KUKA KRL program: Rack_Verde_Inpicker_D.src, Rack_Verde_Inpicker_D.dat

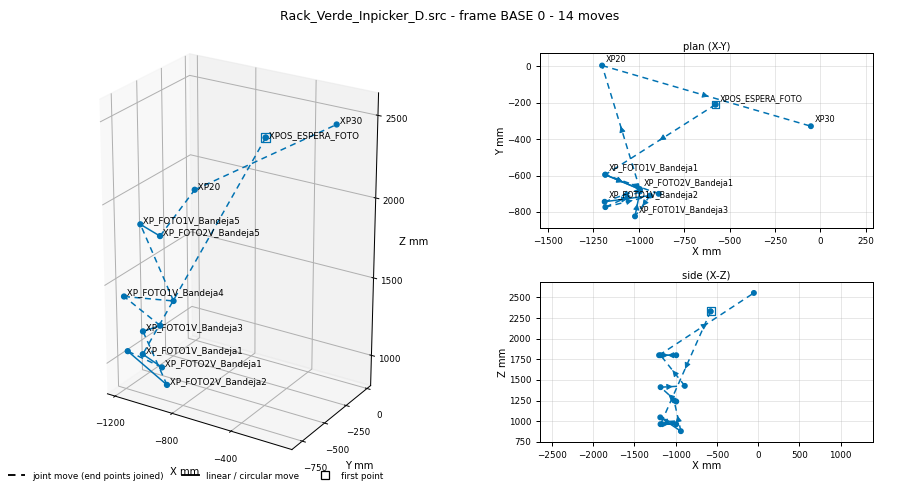
[picture p0: tool path of Rack_Verde_Inpicker_D.src in frame BASE 0, 14 of 14 moves have a stored position in this frame; points joined in program order, loops and branches not executed]
--- Rack_Verde_Inpicker_D.src ---
&ACCESS RVP
&REL 1
&COMMENT FOTOS EN RACK VERDE
&PARAM EDITMASK = *
&PARAM TEMPLATE = C:\KRC\Roboter\Template\vorgabe
&PARAM DISKPATH = KRC:\R1\Program\MAFELEC
DEF Rack_Verde_Inpicker_D( )
;FOLD DECLARACION_INPICKER
DECL EKI_STATUS Ret
DECL INT InPickerStateValue
;ENDFOLD
;FOLD INI;%{PE}
  ;FOLD BASISTECH INI
    GLOBAL INTERRUPT DECL 3 WHEN $STOPMESS==TRUE DO IR_STOPM ( )
    INTERRUPT ON 3
    BAS (#INITMOV,0 )
  ;ENDFOLD (BASISTECH INI)
  ;FOLD USER INI
O_LIMITS_OK=FALSE
O_LIMITS_NOK=FALSE
O_LIMIT_X=FALSE
O_LIMIT_Y=FALSE
O_LIMIT_Z=FALSE
O_LIMIT_A=FALSE
O_LIMIT_B=FALSE
O_LIMIT_C=FALSE
LIM_X=FALSE
LIM_Y=FALSE
LIM_Z=FALSE
LIM_A=FALSE
LIM_B=FALSE
LIM_C=FALSE
O_TYPE_INFO=0

  ;ENDFOLD (USER INI)
;ENDFOLD (INI)

;################################################
; PROYECTO: MAFELEC PLANTA DE BATERIAS
; ROBOT: 121_R1
; PROGRAMA: FOTO PARA CORRECCIONES EN RACK VERDE
; CREADO POR: Alejandro Company(zaisor robotics)
; FECHA: 23-NOVIEMBRE-2022
; MODIFICADO POR:
; FECHA MODIFICACION: 13-ENERO-2023
;################################################

$TIMER[2]=0
$TIMER_STOP[2]=FALSE
;FOLD INICIALIZACION PUERTOS DE KRL
Ret = EKI_INIT("XML_Kuka_InPicker_1")
Ret = EKI_INIT("XML_Kuka_InPicker_2")

Ret = EKI_OPEN("XML_Kuka_InPicker_1")
Ret = EKI_OPEN("XML_Kuka_InPicker_2")

 INPICKER_Handler.DataToSend.command=0
;WAIT FOR (INPICKER_Handler.ConnectionStatus==TRUE)
;IF (INPICKER_Handler.ConnectionStatus==TRUE) THEN
;ELSE
;ENDIF

;ENDFOLD

Empujador(1,"R",FALSE)
Empujador(2,"R",FALSE)

; POSICION DE ESPERA ENTRADA RACK 1
;FOLD PTP POS_ESPERA_FOTO Vel=100 % H Tool[5]:T_Camara Base[0];%{PE}%R 8.3.48,%MKUKATPBASIS,%CMOVE,%VPTP,%P 1:PTP, 2:POS_ESPERA_FOTO, 3:, 5:100, 7:H
$BWDSTART=FALSE
PDAT_ACT=PH
FDAT_ACT=FPOS_ESPERA_FOTO
BAS(#PTP_PARAMS,100)
PTP XPOS_ESPERA_FOTO
;ENDFOLD

;ESPERA AREA 1
WAIT FOR I_ARDY_1
O_AREL_1=FALSE
RV_Bandeja_nr=0

Empujador(1,"R",TRUE)
Empujador(2,"R",TRUE)

;FOLD PTP P11 CONT Vel=100 % M Tool[5]:T_Camara Base[0];%{PE}%R 8.3.48,%MKUKATPBASIS,%CMOVE,%VPTP,%P 1:PTP, 2:P11, 3:C_DIS, 5:100, 7:M
$BWDSTART=FALSE
PDAT_ACT=PM
FDAT_ACT=FP11
BAS(#PTP_PARAMS,100)
PTP XP11 C_DIS
;ENDFOLD

O_TYPE_RQ=TRUE
WAIT FOR (I_TYPE_INFO >= 10) AND (I_TYPE_INFO <= 16)

RV_Bandeja_Nr=I_TYPE_INFO

SWITCH RV_Bandeja_Nr

CASE 11
O_TYPE_RQ=FALSE
O_TYPE_INFO=RV_Bandeja_Nr
INICIO_FOTO1:
;FOLD PTP P_FOTO1V_Bandeja1 Vel=50 % M Tool[5]:T_Camara Base[0];%{PE}%R 8.3.48,%MKUKATPBASIS,%CMOVE,%VPTP,%P 1:PTP, 2:P_FOTO1V_Bandeja1, 3:, 5:50, 7:M
$BWDSTART=FALSE
PDAT_ACT=PM
FDAT_ACT=FP_FOTO1V_Bandeja1
BAS(#PTP_PARAMS,50)
PTP XP_FOTO1V_Bandeja1
;ENDFOLD
;FOLD REALIZA FOTO 1 BANDEJA 1
WAIT SEC 1
Fallo_nr=0
Ini1:
O_INPICKER_OK = FALSE
O_INPICKER_NOK = FALSE
SELECT_SIN=FALSE
SELECT_U1=FALSE
SELECT_U2=FALSE
SELECT_U3=FALSE
SELECT_U4=FALSE

; INICIALIZACION CAMARA PARA BANDEJA 1
 INPICKER_Handler.DataToSend.command=0
 INPICKER_Handler.DataToSend.GraspConfirmation=0
 WAIT FOR (INPICKER_Handler.DataReceived.state==0)

; Camara siempre 2
 INPICKER_Handler.DataToSend.CameraID=2

; contendor igual al numero de bandeja
 INPICKER_Handler.DataToSend.ContainerID=1
 INPICKER_Handler.DataToSend.partid=1
 INPICKER_Handler.DataToSend.GraspConfirmation=0
 WAIT SEC 0.2

; DISPARO FOTO
 INPICKER_Handler.DataToSend.command=1

; ESPERA FOTO REALIZADA
 WAIT FOR (INPICKER_Handler.DataReceived.state==15) OR (INPICKER_Handler.DataReceived.state==-1)

IF (INPICKER_Handler.DataReceived.state==-1) THEN

IF (Fallo_nr>=1) THEN
O_INPICKER_OK=FALSE
O_INPICKER_NOK=TRUE

O_TYPE_RQ = FALSE
WAIT FOR I_TYPE_INFO == 0

O_TYPE_RQ = TRUE
WAIT FOR (I_TYPE_INFO >= 1) AND (I_TYPE_INFO <= 5)

SWITCH I_TYPE_INFO

CASE 2
; #### SELECCION DESDE HMI REINTENTO FOTO ####

SELECT_NEXT=FALSE
O_INPICKER_OK=FALSE
O_INPICKER_NOK=FALSE
O_TYPE_RQ = FALSE
GOTO Ini1

CASE 3
; #### SELECCION DESDE HMI CONT SIN CORRECCION ####

SELECT_SIN=TRUE
O_INPICKER_OK=FALSE
O_INPICKER_NOK=TRUE
O_TYPE_RQ = FALSE
GOTO FIN_FOTO1

CASE 4
; #### SELECCION DESDE HMI CERRAR BANDEJA ####
; #### E IR A SIGUIENTE NIVEL             ####

SELECT_NEXT=TRUE
O_INPICKER_OK=FALSE
O_INPICKER_NOK=FALSE
O_TYPE_RQ = FALSE
GOTO FIN_FOTO1

DEFAULT
ENDSWITCH

ELSE

Fallo_nr=Fallo_nr+1
GOTO Ini1

ENDIF
ENDIF

Fin1:
 WAIT SEC 0.1
;ENDFOLD

INICIO_POS2_B1:
;FOLD LIN P_FOTO2V_Bandeja1 Vel=0.5 m/s M Tool[5]:T_Camara Base[0];%{PE}%R 8.3.48,%MKUKATPBASIS,%CMOVE,%VLIN,%P 1:LIN, 2:P_FOTO2V_Bandeja1, 3:, 5:0.5, 7:M
$BWDSTART=FALSE
LDAT_ACT=LM
FDAT_ACT=FP_FOTO2V_Bandeja1
BAS(#CP_PARAMS,0.5)
LIN XP_FOTO2V_Bandeja1
;ENDFOLD
;FOLD REALIZA FOTO 2 BANDEJA 1 (INFERIOR)
WAIT SEC 1.0
INPICKER_Handler.DataToSend.GraspConfirmation=1

WAIT FOR (INPICKER_Handler.DataReceived.state==30) OR (INPICKER_Handler.dataReceived.state==-1)

WAIT SEC 0.5

INPICKER_Handler.DataToSend.command=0

IF (INPICKER_handler.datareceived.state==30 ) THEN

IF (INPICKER_Handler.DataReceived.ObjectsGraspable>0) THEN

O_INPICKER_OK=TRUE
O_INPICKER_NOK=FALSE

ELSE

O_INPICKER_OK=FALSE
O_INPICKER_NOK=TRUE

ENDIF

ENDIF

IF (INPICKER_handler.datareceived.state==-1 ) OR (INPICKER_Handler.DataReceived.ObjectsGraspable<=0) THEN

O_INPICKER_OK=FALSE
O_INPICKER_NOK=TRUE

O_TYPE_RQ = FALSE
WAIT FOR I_TYPE_INFO == 0

O_TYPE_RQ = TRUE
WAIT FOR (I_TYPE_INFO >= 1) AND (I_TYPE_INFO <= 5)

SWITCH I_TYPE_INFO

CASE 2
; #### SELECCION DESDE HMI REINTENTO FOTO ####

SELECT_NEXT=FALSE
O_INPICKER_OK=FALSE
O_INPICKER_NOK=FALSE
O_TYPE_RQ = FALSE

IF (INPICKER_Handler.DataReceived.ObjectsGraspable>0)THEN
ELSE
GOTO INICIO_FOTO1
ENDIF

WAIT FOR (INPICKER_Handler.DataReceived.state==0)
GOTO INICIO_FOTO1

CASE 3
; #### SELECCION DESDE HMI CONT SIN CORRECCION ####

SELECT_NEXT=FALSE
O_TYPE_RQ = FALSE

CASE 4
; #### SELECCION DESDE HMI CERRAR BANDEJA ####
; #### E IR A SIGUIENTE NIVEL             ####

SELECT_NEXT=TRUE
O_INPICKER_OK=FALSE
O_INPICKER_NOK=FALSE
O_TYPE_RQ = FALSE

DEFAULT
ENDSWITCH

ENDIF
 INPICKER_Handler.DataToSend.command=0

;ENDFOLD
;FOLD ACTUALIZA BASE DE DESCARGA
FRAMEAUX={X 0,Y 0,Z 0,A 0,B 0,C 0}
FRAME_POS={X 0,Y 0,Z 0,A 0,B 0,C 0}

FRAMEAUX=INPICKER_Handler.DataReceived.PartsToGrasp0.Position
FRAME_POS.x=(FRAMEAUX.x/10)
FRAME_POS.y=(FRAMEAUX.y/10)
FRAME_POS.z=(FRAMEAUX.z/10)
FRAME_POS.a=(FRAMEAUX.a/10)
FRAME_POS.b=(FRAMEAUX.b/10)
FRAME_POS.c=(FRAMEAUX.c/10)

IF FRAME_POS.A < 180.0 THEN
FRAME_POS.A = FRAME_POS.A + 360
ENDIF
IF FRAME_POS.B < 180.0 THEN
FRAME_POS.B = FRAME_POS.B + 360
ENDIF
IF FRAME_POS.A > 180.0 THEN
FRAME_POS.A = FRAME_POS.A - 360
ENDIF
IF FRAME_POS.B > 180.0 THEN
FRAME_POS.B = FRAME_POS.B - 360
ENDIF

FRAME_POS.C = FRAME_POS.C - 360

;ENDFOLD
;FOLD CONTROL LIMITES DE VISION
CTRL_limites()
;ENDFOLD
;FOLD DECISION RESULTADOS EVALUACION BANDEJA 1
IF (O_LIMITS_OK==FALSE) AND (O_LIMITS_NOK==TRUE) THEN

O_TYPE_RQ = FALSE
WAIT FOR I_TYPE_INFO == 0

O_TYPE_RQ = TRUE
WAIT FOR (I_TYPE_INFO >= 1) AND (I_TYPE_INFO <= 5)

SWITCH I_TYPE_INFO

CASE 2
; #### SELECCION DESDE HMI REINTENTO FOTO ####

SELECT_NEXT=FALSE
O_TYPE_RQ = FALSE
O_LIMITS_OK = FALSE
O_LIMITS_NOK = FALSE
O_LIMIT_X = FALSE
O_LIMIT_Y = FALSE
O_LIMIT_Z = FALSE
O_LIMIT_A = FALSE
O_LIMIT_B = FALSE
O_LIMIT_C = FALSE

GOTO INICIO_FOTO1

CASE 3
; #### SELECCION DESDE HMI CONT SIN CORRECCION ####

SELECT_NEXT=FALSE
O_TYPE_RQ = FALSE

CASE 4
; #### SELECCION DESDE HMI CERRAR BANDEJA ####
; #### E IR A SIGUIENTE NIVEL             ####

SELECT_NEXT=TRUE
O_TYPE_RQ = FALSE
O_LIMITS_OK = FALSE
O_LIMITS_NOK = FALSE
O_LIMIT_X = FALSE
O_LIMIT_Y = FALSE
O_LIMIT_Z = FALSE
O_LIMIT_A = FALSE
O_LIMIT_B = FALSE
O_LIMIT_C = FALSE

DEFAULT

HALT
HALT
HALT
ENDSWITCH

ENDIF
;ENDFOLD
FIN_FOTO1:

CASE 12
O_TYPE_RQ=FALSE
O_TYPE_INFO=RV_Bandeja_Nr
INICIO_FOTO2:
;FOLD PTP P_FOTO1V_Bandeja2 Vel=50 % M Tool[5]:T_Camara Base[0];%{PE}%R 8.3.48,%MKUKATPBASIS,%CMOVE,%VPTP,%P 1:PTP, 2:P_FOTO1V_Bandeja2, 3:, 5:50, 7:M
$BWDSTART=FALSE
PDAT_ACT=PM
FDAT_ACT=FP_FOTO1V_Bandeja2
BAS(#PTP_PARAMS,50)
PTP XP_FOTO1V_Bandeja2
;ENDFOLD
;FOLD REALIZA FOTO 1 BANDEJA 2
WAIT SEC 1
Fallo_nr=0
Ini2:
O_INPICKER_OK = FALSE
O_INPICKER_NOK = FALSE
SELECT_SIN=FALSE
SELECT_U1=FALSE
SELECT_U2=FALSE
SELECT_U3=FALSE
SELECT_U4=FALSE

; INICIALIZACION CAMARA PARA BANDEJA 2
 INPICKER_Handler.DataToSend.command=0
 INPICKER_Handler.DataToSend.GraspConfirmation=0
 WAIT FOR (INPICKER_Handler.DataReceived.state==0)

; Camara siempre 2
 INPICKER_Handler.DataToSend.CameraID=2

; contendor igual al numero de bandeja
 INPICKER_Handler.DataToSend.ContainerID=2
 INPICKER_Handler.DataToSend.partid=2
 INPICKER_Handler.DataToSend.GraspConfirmation=0
 WAIT SEC 0.2

; DISPARO FOTO
 INPICKER_Handler.DataToSend.command=1

; ESPERA FOTO REALIZADA
 WAIT FOR (INPICKER_Handler.DataReceived.state==15) OR (INPICKER_Handler.DataReceived.state==-1)

IF (INPICKER_Handler.DataReceived.state==-1) THEN

IF (Fallo_nr>=1) THEN
O_INPICKER_OK=FALSE
O_INPICKER_NOK=TRUE

O_TYPE_RQ = FALSE
WAIT FOR I_TYPE_INFO == 0

O_TYPE_RQ = TRUE
WAIT FOR (I_TYPE_INFO >= 1) AND (I_TYPE_INFO <= 5)

SWITCH I_TYPE_INFO

CASE 2
; #### SELECCION DESDE HMI REINTENTO FOTO ####

SELECT_NEXT=FALSE
O_INPICKER_OK=FALSE
O_INPICKER_NOK=FALSE
O_TYPE_RQ = FALSE
GOTO Ini2

CASE 3
; #### SELECCION DESDE HMI CONT SIN CORRECCION ####

SELECT_SIN=TRUE
O_INPICKER_OK=FALSE
O_INPICKER_NOK=TRUE
O_TYPE_RQ = FALSE
GOTO FIN_FOTO2

CASE 4
; #### SELECCION DESDE HMI CERRAR BANDEJA ####
; #### E IR A SIGUIENTE NIVEL             ####

SELECT_NEXT=TRUE
O_INPICKER_OK=FALSE
O_INPICKER_NOK=FALSE
O_TYPE_RQ = FALSE
GOTO FIN_FOTO2

DEFAULT
ENDSWITCH

ELSE

Fallo_nr=Fallo_nr+1
GOTO Ini2

ENDIF
ENDIF

Fin2:
 WAIT SEC 0.1
;ENDFOLD

INICIO_POS2_B2:
;FOLD LIN P_FOTO2V_Bandeja2 Vel=0.5 m/s M Tool[5]:T_Camara Base[0];%{PE}%R 8.3.48,%MKUKATPBASIS,%CMOVE,%VLIN,%P 1:LIN, 2:P_FOTO2V_Bandeja2, 3:, 5:0.5, 7:M
$BWDSTART=FALSE
LDAT_ACT=LM
FDAT_ACT=FP_FOTO2V_Bandeja2
BAS(#CP_PARAMS,0.5)
LIN XP_FOTO2V_Bandeja2
;ENDFOLD
;FOLD REALIZA FOTO 2 BANDEJA 2
WAIT SEC 1.0
INPICKER_Handler.DataToSend.GraspConfirmation=1

WAIT FOR (INPICKER_Handler.DataReceived.state==30) OR (INPICKER_Handler.dataReceived.state==-1)

WAIT SEC 0.5
INPICKER_Handler.DataToSend.command=0

IF (INPICKER_handler.datareceived.state==30 ) THEN

IF (INPICKER_Handler.DataReceived.ObjectsGraspable>0) THEN

O_INPICKER_OK=TRUE
O_INPICKER_NOK=FALSE

ELSE

O_INPICKER_OK=FALSE
O_INPICKER_NOK=TRUE

ENDIF

ENDIF

IF (INPICKER_handler.datareceived.state==-1 ) OR (INPICKER_Handler.DataReceived.ObjectsGraspable<=0) THEN

O_INPICKER_OK=FALSE
O_INPICKER_NOK=TRUE

O_TYPE_RQ = FALSE
WAIT FOR I_TYPE_INFO == 0

O_TYPE_RQ = TRUE
WAIT FOR (I_TYPE_INFO >= 1) AND (I_TYPE_INFO <= 5)

SWITCH I_TYPE_INFO

CASE 2
; #### SELECCION DESDE HMI REINTENTO FOTO ####

SELECT_NEXT=FALSE
O_INPICKER_OK=FALSE
O_INPICKER_NOK=FALSE
O_TYPE_RQ = FALSE

IF (INPICKER_Handler.DataReceived.ObjectsGraspable>0)THEN
ELSE
GOTO INICIO_FOTO2
ENDIF

WAIT FOR (INPICKER_Handler.DataReceived.state==0)
GOTO INICIO_FOTO2

CASE 3
; #### SELECCION DESDE HMI CONT SIN CORRECCION ####

SELECT_NEXT=FALSE
O_TYPE_RQ = FALSE

CASE 4
; #### SELECCION DESDE HMI CERRAR BANDEJA ####
; #### E IR A SIGUIENTE NIVEL             ####

SELECT_NEXT=TRUE
O_INPICKER_OK=FALSE
O_INPICKER_NOK=FALSE
O_TYPE_RQ = FALSE

DEFAULT
ENDSWITCH

ENDIF

 INPICKER_Handler.DataToSend.command=0

;ENDFOLD
;FOLD ACTUALIZA BASE DE DESCARGA
FRAMEAUX={X 0,Y 0,Z 0,A 0,B 0,C 0}
FRAME_POS={X 0,Y 0,Z 0,A 0,B 0,C 0}

FRAMEAUX=INPICKER_Handler.DataReceived.PartsToGrasp0.Position
FRAME_POS.x=(FRAMEAUX.x/10)
FRAME_POS.y=(FRAMEAUX.y/10)
FRAME_POS.z=(FRAMEAUX.z/10)
FRAME_POS.a=(FRAMEAUX.a/10)
FRAME_POS.b=(FRAMEAUX.b/10)
FRAME_POS.c=(FRAMEAUX.c/10)

IF FRAME_POS.A < 180.0 THEN
FRAME_POS.A = FRAME_POS.A + 360
ENDIF

IF FRAME_POS.B < 180.0 THEN
FRAME_POS.B = FRAME_POS.B + 360
ENDIF

IF FRAME_POS.A > 180.0 THEN
FRAME_POS.A = FRAME_POS.A - 360
ENDIF

IF FRAME_POS.B > 180.0 THEN
FRAME_POS.B = FRAME_POS.B - 360
ENDIF

FRAME_POS.C = FRAME_POS.C - 360

;ENDFOLD
;FOLD CONTROL LIMITES DE VISION
CTRL_limites()
;ENDFOLD
;FOLD DECISION RESULTADOS EVALUACION BANDEJA 2
IF (O_LIMITS_OK==FALSE) AND (O_LIMITS_NOK==TRUE) THEN

O_TYPE_RQ = FALSE
WAIT FOR I_TYPE_INFO == 0

O_TYPE_RQ = TRUE
WAIT FOR (I_TYPE_INFO >= 1) AND (I_TYPE_INFO <= 5)

SWITCH I_TYPE_INFO

CASE 2
; #### SELECCION DESDE HMI REINTENTO FOTO ####

SELECT_NEXT=FALSE
O_TYPE_RQ = FALSE
O_LIMITS_OK = FALSE
O_LIMITS_NOK = FALSE
O_LIMIT_X = FALSE
O_LIMIT_Y = FALSE
O_LIMIT_Z = FALSE
O_LIMIT_A = FALSE
O_LIMIT_B = FALSE
O_LIMIT_C = FALSE

GOTO INICIO_FOTO2

CASE 3
; #### SELECCION DESDE HMI CONT SIN CORRECCION ####

SELECT_NEXT=FALSE
O_TYPE_RQ = FALSE

CASE 4
; #### SELECCION DESDE HMI CERRAR BANDEJA ####
; #### E IR A SIGUIENTE NIVEL             ####

SELECT_NEXT=TRUE
O_TYPE_RQ = FALSE
O_LIMITS_OK = FALSE
O_LIMITS_NOK = FALSE
O_LIMIT_X = FALSE
O_LIMIT_Y = FALSE
O_LIMIT_Z = FALSE
O_LIMIT_A = FALSE
O_LIMIT_B = FALSE
O_LIMIT_C = FALSE

DEFAULT

HALT
HALT
HALT
ENDSWITCH

ENDIF
;ENDFOLD
FIN_FOTO2:

CASE 13
O_TYPE_RQ=FALSE
O_TYPE_INFO=RV_Bandeja_Nr
INICIO_FOTO3:
;FOLD PTP P_FOTO1V_Bandeja3 Vel=50 % M Tool[5]:T_Camara Base[0];%{PE}%R 8.3.48,%MKUKATPBASIS,%CMOVE,%VPTP,%P 1:PTP, 2:P_FOTO1V_Bandeja3, 3:, 5:50, 7:M
$BWDSTART=FALSE
PDAT_ACT=PM
FDAT_ACT=FP_FOTO1V_Bandeja3
BAS(#PTP_PARAMS,50)
PTP XP_FOTO1V_Bandeja3
;ENDFOLD
;FOLD REALIZA FOTO 1 BANDEJA 1
WAIT SEC 1
Fallo_nr=0
Ini3:
O_INPICKER_OK = FALSE
O_INPICKER_NOK = FALSE
SELECT_SIN=FALSE
SELECT_U1=FALSE
SELECT_U2=FALSE
SELECT_U3=FALSE
SELECT_U4=FALSE

; INICIALIZACION CAMARA PARA BANDEJA 3
 INPICKER_Handler.DataToSend.command=0
 INPICKER_Handler.DataToSend.GraspConfirmation=0
 WAIT FOR (INPICKER_Handler.DataReceived.state==0)

; Camara siempre 2
 INPICKER_Handler.DataToSend.CameraID=2

; contendor igual al numero de bandeja
 INPICKER_Handler.DataToSend.ContainerID=3
 INPICKER_Handler.DataToSend.partid=3
 INPICKER_Handler.DataToSend.GraspConfirmation=0
 WAIT SEC 0.2

; DISPARO FOTO
 INPICKER_Handler.DataToSend.command=1

; ESPERA FOTO REALIZADA
 WAIT FOR (INPICKER_Handler.DataReceived.state==15) OR (INPICKER_Handler.DataReceived.state==-1)

IF (INPICKER_Handler.DataReceived.state==-1) THEN

IF (Fallo_nr>=1) THEN
O_INPICKER_OK=FALSE
O_INPICKER_NOK=TRUE

O_TYPE_RQ = FALSE
WAIT FOR I_TYPE_INFO == 0

O_TYPE_RQ = TRUE
WAIT FOR (I_TYPE_INFO >= 1) AND (I_TYPE_INFO <= 5)

SWITCH I_TYPE_INFO

CASE 2
; #### SELECCION DESDE HMI REINTENTO FOTO ####

SELECT_NEXT=FALSE
O_INPICKER_OK=FALSE
O_INPICKER_NOK=FALSE
O_TYPE_RQ = FALSE
GOTO Ini3

CASE 3
; #### SELECCION DESDE HMI CONT SIN CORRECCION ####

SELECT_SIN=TRUE
O_INPICKER_OK=FALSE
O_INPICKER_NOK=TRUE
O_TYPE_RQ = FALSE
GOTO FIN_FOTO3

CASE 4
; #### SELECCION DESDE HMI CERRAR BANDEJA ####
; #### E IR A SIGUIENTE NIVEL             ####

SELECT_NEXT=TRUE
O_INPICKER_OK=FALSE
O_INPICKER_NOK=FALSE
O_TYPE_RQ = FALSE
GOTO FIN_FOTO3

DEFAULT
ENDSWITCH

ELSE

Fallo_nr=Fallo_nr+1
GOTO Ini3

ENDIF
ENDIF

Fin3:
 WAIT SEC 0.1
;ENDFOLD

INICIO_POS2_B3:
;FOLD LIN P_FOTO2V_Bandeja3 Vel=0.3 m/s M Tool[5]:T_Camara Base[0];%{PE}%R 8.3.48,%MKUKATPBASIS,%CMOVE,%VLIN,%P 1:LIN, 2:P_FOTO2V_Bandeja3, 3:, 5:0.3, 7:M
$BWDSTART=FALSE
LDAT_ACT=LM
FDAT_ACT=FP_FOTO2V_Bandeja3
BAS(#CP_PARAMS,0.3)
LIN XP_FOTO2V_Bandeja3
;ENDFOLD
;FOLD REALIZA FOTO 2 BANDEJA 3
WAIT SEC 1.0
INPICKER_Handler.DataToSend.GraspConfirmation=1

WAIT FOR (INPICKER_Handler.DataReceived.state==30) OR (INPICKER_Handler.dataReceived.state==-1)

WAIT SEC 0.5

INPICKER_Handler.DataToSend.command=0

IF (INPICKER_handler.datareceived.state==30 ) THEN

IF (INPICKER_Handler.DataReceived.ObjectsGraspable>0) THEN

O_INPICKER_OK=TRUE
O_INPICKER_NOK=FALSE

ELSE

O_INPICKER_OK=FALSE
O_INPICKER_NOK=TRUE

ENDIF

ENDIF

IF (INPICKER_handler.datareceived.state==-1 ) OR (INPICKER_Handler.DataReceived.ObjectsGraspable<=0) THEN

O_INPICKER_OK=FALSE
O_INPICKER_NOK=TRUE

O_TYPE_RQ = FALSE
WAIT FOR I_TYPE_INFO == 0

O_TYPE_RQ = TRUE
WAIT FOR (I_TYPE_INFO >= 1) AND (I_TYPE_INFO <= 5)

SWITCH I_TYPE_INFO

CASE 2
; #### SELECCION DESDE HMI REINTENTO FOTO ####

SELECT_NEXT=FALSE
O_INPICKER_OK=FALSE
O_INPICKER_NOK=FALSE
O_TYPE_RQ = FALSE

IF (INPICKER_Handler.DataReceived.ObjectsGraspable>0)THEN
ELSE
GOTO INICIO_FOTO3
ENDIF

WAIT FOR (INPICKER_Handler.DataReceived.state==0)
GOTO INICIO_FOTO3

CASE 3
; #### SELECCION DESDE HMI CONT SIN CORRECCION ####

SELECT_NEXT=FALSE
O_TYPE_RQ = FALSE

CASE 4
; #### SELECCION DESDE HMI CERRAR BANDEJA ####
; #### E IR A SIGUIENTE NIVEL             ####

SELECT_NEXT=TRUE
O_INPICKER_OK=FALSE
O_INPICKER_NOK=FALSE
O_TYPE_RQ = FALSE

DEFAULT
ENDSWITCH

ENDIF
 INPICKER_Handler.DataToSend.command=0

;ENDFOLD
;FOLD ACTUALIZA BASE DE DESCARGA
FRAMEAUX={X 0,Y 0,Z 0,A 0,B 0,C 0}
FRAME_POS={X 0,Y 0,Z 0,A 0,B 0,C 0}

FRAMEAUX=INPICKER_Handler.DataReceived.PartsToGrasp0.Position
FRAME_POS.x=(FRAMEAUX.x/10)
FRAME_POS.y=(FRAMEAUX.y/10)
FRAME_POS.z=(FRAMEAUX.z/10)
FRAME_POS.a=(FRAMEAUX.a/10)
FRAME_POS.b=(FRAMEAUX.b/10)
FRAME_POS.c=(FRAMEAUX.c/10)

IF FRAME_POS.A < 180.0 THEN
FRAME_POS.A = FRAME_POS.A + 360
ENDIF

IF FRAME_POS.B < 180.0 THEN
FRAME_POS.B = FRAME_POS.B + 360
ENDIF

IF FRAME_POS.A > 180.0 THEN
FRAME_POS.A = FRAME_POS.A - 360
ENDIF

IF FRAME_POS.B > 180.0 THEN
FRAME_POS.B = FRAME_POS.B - 360
ENDIF

FRAME_POS.C = FRAME_POS.C - 360

;ENDFOLD
;FOLD CONTROL LIMITES DE VISION
CTRL_limites()
;ENDFOLD
;FOLD DECISION RESULTADOS EVALUACION BANDEJA 3
IF (O_LIMITS_OK==FALSE) AND (O_LIMITS_NOK==TRUE) THEN

O_TYPE_RQ = FALSE
WAIT FOR I_TYPE_INFO == 0

O_TYPE_RQ = TRUE
WAIT FOR (I_TYPE_INFO >= 1) AND (I_TYPE_INFO <= 5)

SWITCH I_TYPE_INFO

CASE 2
; #### SELECCION DESDE HMI REINTENTO FOTO ####

SELECT_NEXT=FALSE
O_TYPE_RQ = FALSE
O_LIMITS_OK = FALSE
O_LIMITS_NOK = FALSE
O_LIMIT_X = FALSE
O_LIMIT_Y = FALSE
O_LIMIT_Z = FALSE
O_LIMIT_A = FALSE
O_LIMIT_B = FALSE
O_LIMIT_C = FALSE

GOTO INICIO_FOTO3

CASE 3
; #### SELECCION DESDE HMI CONT SIN CORRECCION ####

SELECT_NEXT=FALSE
O_TYPE_RQ = FALSE

CASE 4
; #### SELECCION DESDE HMI CERRAR BANDEJA ####
; #### E IR A SIGUIENTE NIVEL             ####

SELECT_NEXT=TRUE
O_TYPE_RQ = FALSE
O_LIMITS_OK = FALSE
O_LIMITS_NOK = FALSE
O_LIMIT_X = FALSE
O_LIMIT_Y = FALSE
O_LIMIT_Z = FALSE
O_LIMIT_A = FALSE
O_LIMIT_B = FALSE
O_LIMIT_C = FALSE

DEFAULT

HALT
HALT
HALT
ENDSWITCH

ENDIF
;ENDFOLD
FIN_FOTO3:

CASE 14
O_TYPE_RQ=FALSE
O_TYPE_INFO=RV_Bandeja_Nr
INICIO_FOTO4:
;FOLD PTP P_FOTO1V_Bandeja4 Vel=50 % M Tool[5]:T_Camara Base[0];%{PE}%R 8.3.48,%MKUKATPBASIS,%CMOVE,%VPTP,%P 1:PTP, 2:P_FOTO1V_Bandeja4, 3:, 5:50, 7:M
$BWDSTART=FALSE
PDAT_ACT=PM
FDAT_ACT=FP_FOTO1V_Bandeja4
BAS(#PTP_PARAMS,50)
PTP XP_FOTO1V_Bandeja4
;ENDFOLD
;FOLD REALIZA FOTO 1 BANDEJA 4
WAIT SEC 1
Fallo_nr=0
Ini4:
O_INPICKER_OK = FALSE
O_INPICKER_NOK = FALSE
SELECT_SIN=FALSE
SELECT_U1=FALSE
SELECT_U2=FALSE
SELECT_U3=FALSE
SELECT_U4=FALSE

; INICIALIZACION CAMARA PARA BANDEJA 4
 INPICKER_Handler.DataToSend.command=0
 INPICKER_Handler.DataToSend.GraspConfirmation=0
 WAIT FOR (INPICKER_Handler.DataReceived.state==0)

; Camara siempre 2
 INPICKER_Handler.DataToSend.CameraID=2

; contendor igual al numero de bandeja
 INPICKER_Handler.DataToSend.ContainerID=4
 INPICKER_Handler.DataToSend.partid=4
 INPICKER_Handler.DataToSend.GraspConfirmation=0
 WAIT SEC 0.2

; DISPARO FOTO
 INPICKER_Handler.DataToSend.command=1

; ESPERA FOTO REALIZADA
 WAIT FOR (INPICKER_Handler.DataReceived.state==15) OR (INPICKER_Handler.DataReceived.state==-1)

IF (INPICKER_Handler.DataReceived.state==-1) THEN

IF (Fallo_nr>=1) THEN
O_INPICKER_OK=FALSE
O_INPICKER_NOK=TRUE

O_TYPE_RQ = FALSE
WAIT FOR I_TYPE_INFO == 0

O_TYPE_RQ = TRUE
WAIT FOR (I_TYPE_INFO >= 1) AND (I_TYPE_INFO <= 5)

SWITCH I_TYPE_INFO

CASE 2
; #### SELECCION DESDE HMI REINTENTO FOTO ####

SELECT_NEXT=FALSE
O_INPICKER_OK=FALSE
O_INPICKER_NOK=FALSE
O_TYPE_RQ = FALSE
GOTO Ini4

CASE 3
; #### SELECCION DESDE HMI CONT SIN CORRECCION ####

SELECT_SIN=TRUE
O_INPICKER_OK=FALSE
O_INPICKER_NOK=TRUE
O_TYPE_RQ = FALSE
GOTO FIN_FOTO4

CASE 4
; #### SELECCION DESDE HMI CERRAR BANDEJA ####
; #### E IR A SIGUIENTE NIVEL             ####

SELECT_NEXT=TRUE
O_INPICKER_OK=FALSE
O_INPICKER_NOK=FALSE
O_TYPE_RQ = FALSE
GOTO FIN_FOTO4

DEFAULT
ENDSWITCH

ELSE

Fallo_nr=Fallo_nr+1
GOTO Ini4

ENDIF
ENDIF

Fin4:
 WAIT SEC 0.1
;ENDFOLD

INICIO_POS2_B4:
;FOLD PTP P_FOTO2V_Bandeja4 Vel=50 % M Tool[5]:T_Camara Base[0];%{PE}%R 8.3.48,%MKUKATPBASIS,%CMOVE,%VPTP,%P 1:PTP, 2:P_FOTO2V_Bandeja4, 3:, 5:50, 7:M
$BWDSTART=FALSE
PDAT_ACT=PM
FDAT_ACT=FP_FOTO2V_Bandeja4
BAS(#PTP_PARAMS,50)
PTP XP_FOTO2V_Bandeja4
;ENDFOLD
;FOLD REALIZA FOTO 2 BANDEJA 4
WAIT SEC 1.0
INPICKER_Handler.DataToSend.GraspConfirmation=1

WAIT FOR (INPICKER_Handler.DataReceived.state==30) OR (INPICKER_Handler.dataReceived.state==-1)

WAIT SEC 0.5

INPICKER_Handler.DataToSend.command=0

IF (INPICKER_handler.datareceived.state==30 ) THEN

IF (INPICKER_Handler.DataReceived.ObjectsGraspable>0) THEN

O_INPICKER_OK=TRUE
O_INPICKER_NOK=FALSE

ELSE

O_INPICKER_OK=FALSE
O_INPICKER_NOK=TRUE

ENDIF

ENDIF

IF (INPICKER_handler.datareceived.state==-1 ) OR (INPICKER_Handler.DataReceived.ObjectsGraspable<=0) THEN

O_INPICKER_OK=FALSE
O_INPICKER_NOK=TRUE

O_TYPE_RQ = FALSE
WAIT FOR I_TYPE_INFO == 0

O_TYPE_RQ = TRUE
WAIT FOR (I_TYPE_INFO >= 1) AND (I_TYPE_INFO <= 5)

SWITCH I_TYPE_INFO

CASE 2
; #### SELECCION DESDE HMI REINTENTO FOTO ####

SELECT_NEXT=FALSE
O_INPICKER_OK=FALSE
O_INPICKER_NOK=FALSE
O_TYPE_RQ = FALSE

IF (INPICKER_Handler.DataReceived.ObjectsGraspable>0)THEN
ELSE
GOTO INICIO_FOTO4
ENDIF

WAIT FOR (INPICKER_Handler.DataReceived.state==0)
GOTO INICIO_FOTO4

CASE 3
; #### SELECCION DESDE HMI CONT SIN CORRECCION ####

SELECT_NEXT=FALSE
O_TYPE_RQ = FALSE

CASE 4
; #### SELECCION DESDE HMI CERRAR BANDEJA ####
; #### E IR A SIGUIENTE NIVEL             ####

SELECT_NEXT=TRUE
O_INPICKER_OK=FALSE
O_INPICKER_NOK=FALSE
O_TYPE_RQ = FALSE

DEFAULT
ENDSWITCH

ENDIF
 INPICKER_Handler.DataToSend.command=0

;ENDFOLD
;FOLD ACTUALIZA BASE DE DESCARGA
FRAMEAUX={X 0,Y 0,Z 0,A 0,B 0,C 0}
FRAME_POS={X 0,Y 0,Z 0,A 0,B 0,C 0}

FRAMEAUX=INPICKER_Handler.DataReceived.PartsToGrasp0.Position
FRAME_POS.x=(FRAMEAUX.x/10)
FRAME_POS.y=(FRAMEAUX.y/10)
FRAME_POS.z=(FRAMEAUX.z/10)
FRAME_POS.a=(FRAMEAUX.a/10)
FRAME_POS.b=(FRAMEAUX.b/10)
FRAME_POS.c=(FRAMEAUX.c/10)

IF FRAME_POS.A < 180.0 THEN
FRAME_POS.A = FRAME_POS.A + 360
ENDIF
IF FRAME_POS.B < 180.0 THEN
FRAME_POS.B = FRAME_POS.B + 360
ENDIF
IF FRAME_POS.A > 180.0 THEN
FRAME_POS.A = FRAME_POS.A - 360
ENDIF
IF FRAME_POS.B > 180.0 THEN
FRAME_POS.B = FRAME_POS.B - 360
ENDIF

FRAME_POS.C = FRAME_POS.C - 360

;ENDFOLD
;FOLD CONTROL LIMITES DE VISION
CTRL_limites()
;ENDFOLD
;FOLD DECISION RESULTADOS EVALUACION BANDEJA 4
IF (O_LIMITS_OK==FALSE) AND (O_LIMITS_NOK==TRUE) THEN

O_TYPE_RQ = FALSE
WAIT FOR I_TYPE_INFO == 0

O_TYPE_RQ = TRUE
WAIT FOR (I_TYPE_INFO >= 1) AND (I_TYPE_INFO <= 5)

SWITCH I_TYPE_INFO

CASE 2
; #### SELECCION DESDE HMI REINTENTO FOTO ####

SELECT_NEXT=FALSE
O_TYPE_RQ = FALSE
O_LIMITS_OK = FALSE
O_LIMITS_NOK = FALSE
O_LIMIT_X = FALSE
O_LIMIT_Y = FALSE
O_LIMIT_Z = FALSE
O_LIMIT_A = FALSE
O_LIMIT_B = FALSE
O_LIMIT_C = FALSE

GOTO INICIO_FOTO4

CASE 3
; #### SELECCION DESDE HMI CONT SIN CORRECCION ####

SELECT_NEXT=FALSE
O_TYPE_RQ = FALSE

CASE 4
; #### SELECCION DESDE HMI CERRAR BANDEJA ####
; #### E IR A SIGUIENTE NIVEL             ####

SELECT_NEXT=TRUE
O_TYPE_RQ = FALSE
O_LIMITS_OK = FALSE
O_LIMITS_NOK = FALSE
O_LIMIT_X = FALSE
O_LIMIT_Y = FALSE
O_LIMIT_Z = FALSE
O_LIMIT_A = FALSE
O_LIMIT_B = FALSE
O_LIMIT_C = FALSE

DEFAULT

HALT
HALT
HALT
ENDSWITCH

ENDIF
;ENDFOLD
FIN_FOTO4:

CASE 15
O_TYPE_RQ=FALSE
O_TYPE_INFO=RV_Bandeja_Nr
INICIO_FOTO5:
;FOLD PTP P_FOTO1V_Bandeja5 Vel=50 % M Tool[5]:T_Camara Base[0];%{PE}%R 8.3.48,%MKUKATPBASIS,%CMOVE,%VPTP,%P 1:PTP, 2:P_FOTO1V_Bandeja5, 3:, 5:50, 7:M
$BWDSTART=FALSE
PDAT_ACT=PM
FDAT_ACT=FP_FOTO1V_Bandeja5
BAS(#PTP_PARAMS,50)
PTP XP_FOTO1V_Bandeja5
;ENDFOLD
;FOLD REALIZA FOTO 1 BANDEJA 5
WAIT SEC 1
Fallo_nr=0
Ini5:
O_INPICKER_OK = FALSE
O_INPICKER_NOK = FALSE
SELECT_SIN=FALSE
SELECT_U1=FALSE
SELECT_U2=FALSE
SELECT_U3=FALSE
SELECT_U4=FALSE

; INICIALIZACION CAMARA PARA BANDEJA 5
 INPICKER_Handler.DataToSend.command=0
 INPICKER_Handler.DataToSend.GraspConfirmation=0
 WAIT FOR (INPICKER_Handler.DataReceived.state==0)

; Camara siempre 2
 INPICKER_Handler.DataToSend.CameraID=2

; contendor igual al numero de bandeja
 INPICKER_Handler.DataToSend.ContainerID=5
 INPICKER_Handler.DataToSend.partid=5
 INPICKER_Handler.DataToSend.GraspConfirmation=0
 WAIT SEC 0.2

; DISPARO FOTO
 INPICKER_Handler.DataToSend.command=1

; ESPERA FOTO REALIZADA
 WAIT FOR (INPICKER_Handler.DataReceived.state==15) OR (INPICKER_Handler.DataReceived.state==-1)

IF (INPICKER_Handler.DataReceived.state==-1) THEN

IF (Fallo_nr>=1) THEN
O_INPICKER_OK=FALSE
O_INPICKER_NOK=TRUE

O_TYPE_RQ = FALSE
WAIT FOR I_TYPE_INFO == 0

O_TYPE_RQ = TRUE
WAIT FOR (I_TYPE_INFO >= 1) AND (I_TYPE_INFO <= 5)

SWITCH I_TYPE_INFO

CASE 2
; #### SELECCION DESDE HMI REINTENTO FOTO ####

SELECT_NEXT=FALSE
O_INPICKER_OK=FALSE
O_INPICKER_NOK=FALSE
O_TYPE_RQ = FALSE
GOTO Ini5

CASE 3
; #### SELECCION DESDE HMI CONT SIN CORRECCION ####

SELECT_SIN=TRUE
O_INPICKER_OK=FALSE
O_INPICKER_NOK=TRUE
O_TYPE_RQ = FALSE
GOTO FIN_FOTO5

CASE 4
; #### SELECCION DESDE HMI CERRAR BANDEJA ####
; #### E IR A SIGUIENTE NIVEL             ####

SELECT_NEXT=TRUE
O_INPICKER_OK=FALSE
O_INPICKER_NOK=FALSE
O_TYPE_RQ = FALSE
GOTO FIN_FOTO5

DEFAULT
ENDSWITCH

ELSE

Fallo_nr=Fallo_nr+1
GOTO Ini5

ENDIF
ENDIF

Fin5:
 WAIT SEC 0.1
;ENDFOLD

INICIO_POS2_B5:
;FOLD LIN P_FOTO2V_Bandeja5 Vel=0.5 m/s M Tool[5]:T_Camara Base[0];%{PE}%R 8.3.48,%MKUKATPBASIS,%CMOVE,%VLIN,%P 1:LIN, 2:P_FOTO2V_Bandeja5, 3:, 5:0.5, 7:M
$BWDSTART=FALSE
LDAT_ACT=LM
FDAT_ACT=FP_FOTO2V_Bandeja5
BAS(#CP_PARAMS,0.5)
LIN XP_FOTO2V_Bandeja5
;ENDFOLD
;FOLD REALIZA FOTO 2 BANDEJA 5
WAIT SEC 1.0
INPICKER_Handler.DataToSend.GraspConfirmation=1

WAIT FOR (INPICKER_Handler.DataReceived.state==30) OR (INPICKER_Handler.dataReceived.state==-1)

WAIT SEC 0.5

INPICKER_Handler.DataToSend.command=0

IF (INPICKER_handler.datareceived.state==30 ) THEN

IF (INPICKER_Handler.DataReceived.ObjectsGraspable>0) THEN

O_INPICKER_OK=TRUE
O_INPICKER_NOK=FALSE

ELSE

O_INPICKER_OK=FALSE
O_INPICKER_NOK=TRUE

ENDIF

ENDIF

IF (INPICKER_handler.datareceived.state==-1 ) OR (INPICKER_Handler.DataReceived.ObjectsGraspable<=0) THEN

O_INPICKER_OK=FALSE
O_INPICKER_NOK=TRUE

O_TYPE_RQ = FALSE
WAIT FOR I_TYPE_INFO == 0

O_TYPE_RQ = TRUE
WAIT FOR (I_TYPE_INFO >= 1) AND (I_TYPE_INFO <= 5)

SWITCH I_TYPE_INFO

CASE 2
; #### SELECCION DESDE HMI REINTENTO FOTO ####

SELECT_NEXT=FALSE
O_INPICKER_OK=FALSE
O_INPICKER_NOK=FALSE
O_TYPE_RQ = FALSE

IF (INPICKER_Handler.DataReceived.ObjectsGraspable>0)THEN
ELSE
GOTO INICIO_FOTO5
ENDIF

WAIT FOR (INPICKER_Handler.DataReceived.state==0)
GOTO INICIO_FOTO5

CASE 3
; #### SELECCION DESDE HMI CONT SIN CORRECCION ####

SELECT_NEXT=FALSE
O_TYPE_RQ = FALSE

CASE 4
; #### SELECCION DESDE HMI CERRAR BANDEJA ####
; #### E IR A SIGUIENTE NIVEL             ####

SELECT_NEXT=TRUE
O_INPICKER_OK=FALSE
O_INPICKER_NOK=FALSE
O_TYPE_RQ = FALSE

DEFAULT
ENDSWITCH

ENDIF
 INPICKER_Handler.DataToSend.command=0

;ENDFOLD
;FOLD ACTUALIZA BASE DE DESCARGA
FRAMEAUX={X 0,Y 0,Z 0,A 0,B 0,C 0}
FRAME_POS={X 0,Y 0,Z 0,A 0,B 0,C 0}

FRAMEAUX=INPICKER_Handler.DataReceived.PartsToGrasp0.Position
FRAME_POS.x=(FRAMEAUX.x/10)
FRAME_POS.y=(FRAMEAUX.y/10)
FRAME_POS.z=(FRAMEAUX.z/10)
FRAME_POS.a=(FRAMEAUX.a/10)
FRAME_POS.b=(FRAMEAUX.b/10)
FRAME_POS.c=(FRAMEAUX.c/10)

IF FRAME_POS.A < 180.0 THEN
FRAME_POS.A = FRAME_POS.A + 360
ENDIF
IF FRAME_POS.B < 180.0 THEN
FRAME_POS.B = FRAME_POS.B + 360
ENDIF
IF FRAME_POS.A > 180.0 THEN
FRAME_POS.A = FRAME_POS.A - 360
ENDIF
IF FRAME_POS.B > 180.0 THEN
FRAME_POS.B = FRAME_POS.B - 360
ENDIF

FRAME_POS.C = FRAME_POS.C - 360

;ENDFOLD
;FOLD CONTROL LIMITES DE VISION
CTRL_limites()
;ENDFOLD
;FOLD DECISION RESULTADOS EVALUACION BANDEJA 5
IF (O_LIMITS_OK==FALSE) AND (O_LIMITS_NOK==TRUE) THEN

O_TYPE_RQ = FALSE
WAIT FOR I_TYPE_INFO == 0

O_TYPE_RQ = TRUE
WAIT FOR (I_TYPE_INFO >= 1) AND (I_TYPE_INFO <= 5)

SWITCH I_TYPE_INFO

CASE 2
; #### SELECCION DESDE HMI REINTENTO FOTO ####

SELECT_NEXT=FALSE
O_TYPE_RQ = FALSE
O_LIMITS_OK = FALSE
O_LIMITS_NOK = FALSE
O_LIMIT_X = FALSE
O_LIMIT_Y = FALSE
O_LIMIT_Z = FALSE
O_LIMIT_A = FALSE
O_LIMIT_B = FALSE
O_LIMIT_C = FALSE

GOTO INICIO_FOTO5

CASE 3
; #### SELECCION DESDE HMI CONT SIN CORRECCION ####

SELECT_NEXT=FALSE
O_TYPE_RQ = FALSE

CASE 4
; #### SELECCION DESDE HMI CERRAR BANDEJA ####
; #### E IR A SIGUIENTE NIVEL             ####

SELECT_NEXT=TRUE
O_TYPE_RQ = FALSE
O_LIMITS_OK = FALSE
O_LIMITS_NOK = FALSE
O_LIMIT_X = FALSE
O_LIMIT_Y = FALSE
O_LIMIT_Z = FALSE
O_LIMIT_A = FALSE
O_LIMIT_B = FALSE
O_LIMIT_C = FALSE

DEFAULT

HALT
HALT
HALT
ENDSWITCH

ENDIF
;ENDFOLD
FIN_FOTO5:

DEFAULT
ENDSWITCH

FIN:

;FOLD PTP P20 CONT Vel=100 % H Tool[5]:T_Camara Base[0];%{PE}%R 8.3.48,%MKUKATPBASIS,%CMOVE,%VPTP,%P 1:PTP, 2:P20, 3:C_DIS, 5:100, 7:H
$BWDSTART=FALSE
PDAT_ACT=PH
FDAT_ACT=FP20
BAS(#PTP_PARAMS,100)
PTP XP20 C_DIS
;ENDFOLD

IF (SELECT_NEXT == TRUE) THEN

Rack_Verde_Cerrar_D()

ELSE

;FOLD PTP P30 Vel=100 % H Tool[5]:T_Camara Base[0];%{PE}%R 8.3.48,%MKUKATPBASIS,%CMOVE,%VPTP,%P 1:PTP, 2:P30, 3:, 5:100, 7:H
$BWDSTART=FALSE
PDAT_ACT=PH
FDAT_ACT=FP30
BAS(#PTP_PARAMS,100)
PTP XP30
;ENDFOLD

; POSICION DE SALIDA RACK 1
O_AREL_1=TRUE
ENDIF

$TIMER_STOP[2]=TRUE
END
DEF CTRL_limites ()
;################################################
; RUTINA DE CONTROL DE LIMITES DE VISION
;
;################################################

IF $T1 THEN
O_LIMITS_OK=FALSE
O_LIMITS_NOK=FALSE
O_LIMIT_X=FALSE
O_LIMIT_Y=FALSE
O_LIMIT_Z=FALSE
O_LIMIT_A=FALSE
O_LIMIT_B=FALSE
O_LIMIT_C=FALSE

LIM_X=FALSE
LIM_Y=FALSE
LIM_Z=FALSE
LIM_A=FALSE
LIM_B=FALSE
LIM_C=FALSE

ELSE

WAIT FOR $EXT
O_LIMITS_OK=FALSE
O_LIMITS_NOK=FALSE
O_LIMIT_X=FALSE
O_LIMIT_Y=FALSE
O_LIMIT_Z=FALSE
O_LIMIT_A=FALSE
O_LIMIT_B=FALSE
O_LIMIT_C=FALSE

LIM_X=FALSE
LIM_Y=FALSE
LIM_Z=FALSE
LIM_A=FALSE
LIM_B=FALSE
LIM_C=FALSE

IF (FRAME_POS.X>-1000.0) AND (FRAME_POS.X<-970.0) THEN
O_LIMIT_X=TRUE
LIM_X=TRUE
ELSE
O_LIMIT_X=FALSE
LIM_X=FALSE
ENDIF

IF (FRAME_POS.Y>-1690.0) AND (FRAME_POS.Y<-1620.0) THEN
O_LIMIT_Y=TRUE
LIM_Y=TRUE
ELSE
O_LIMIT_Y=FALSE
LIM_Y=FALSE
ENDIF

SWITCH RV_Bandeja_Nr
CASE 11
IF (FRAME_POS.Z>150.0) AND (FRAME_POS.Z<180.0) THEN
O_LIMIT_Z=TRUE
LIM_Z=TRUE
ELSE
O_LIMIT_Z=FALSE
LIM_Z=FALSE
ENDIF
CASE 12
IF (FRAME_POS.Z>350.0) AND (FRAME_POS.Z<380.0) THEN
O_LIMIT_Z=TRUE
LIM_Z=TRUE
ELSE
O_LIMIT_Z=FALSE
LIM_Z=FALSE
ENDIF
CASE 13
IF (FRAME_POS.Z>560.0) AND (FRAME_POS.Z<585.0) THEN
O_LIMIT_Z=TRUE
LIM_Z=TRUE
ELSE
O_LIMIT_Z=FALSE
LIM_Z=FALSE
ENDIF
CASE 14
IF (FRAME_POS.Z>770.0) AND (FRAME_POS.Z<790.0) THEN
O_LIMIT_Z=TRUE
LIM_Z=TRUE
ELSE
O_LIMIT_Z=FALSE
LIM_Z=FALSE
ENDIF
CASE 15
IF (FRAME_POS.Z>970.0) AND (FRAME_POS.Z<1010.0) THEN
O_LIMIT_Z=TRUE
LIM_Z=TRUE
ELSE
O_LIMIT_Z=FALSE
LIM_Z=FALSE
ENDIF
DEFAULT
ENDSWITCH

IF (FRAME_POS.A>-91.30) AND (FRAME_POS.A<-89.50) THEN
O_LIMIT_A=TRUE
LIM_A=TRUE
ELSE
O_LIMIT_A=FALSE
LIM_A=FALSE
ENDIF

IF (FRAME_POS.B>-1.35) AND (FRAME_POS.B<0.75) THEN
O_LIMIT_B=TRUE
LIM_B=TRUE
ELSE
O_LIMIT_B=FALSE
LIM_B=FALSE
ENDIF

IF (FRAME_POS.C>-180.5) AND (FRAME_POS.C<-179.0) THEN
O_LIMIT_C=TRUE
LIM_C=TRUE
ELSE
O_LIMIT_C=FALSE
LIM_A=FALSE
ENDIF

IF (LIM_X==TRUE) AND (LIM_Y==TRUE) AND (LIM_Z==TRUE) AND (LIM_A==TRUE) AND (LIM_B==TRUE) AND (LIM_C==TRUE) THEN
O_LIMITS_OK=TRUE
O_LIMITS_NOK=FALSE
ELSE
O_LIMITS_OK=FALSE
O_LIMITS_NOK=TRUE
ENDIF

;################################################
ENDIF
END

--- Rack_Verde_Inpicker_D.dat ---
&ACCESS RVP
&REL 1
&COMMENT FOTOS EN RACK VERDE
&PARAM EDITMASK = *
&PARAM TEMPLATE = C:\KRC\Roboter\Template\vorgabe
&PARAM DISKPATH = KRC:\R1\Program\MAFELEC
DEFDAT Rack_Verde_Inpicker_D
;FOLD EXTERNAL DECLARATIONS;%{PE}%MKUKATPBASIS,%CEXT,%VCOMMON,%P
;FOLD GRIPPERTECH EXT
EXT  H50 (INT  :IN,INT  :IN,INT  :IN,GRP_TYP  :IN )
;ENDFOLD (GRIPPERTECH EXT)
;FOLD SPOTTECH EXT
EXT  USERSPOT (S_COMMAND  :IN,SPOT_TYPE  :IN )
;ENDFOLD (SPOTTECH EXT)
;FOLD BASISTECH EXT;%{PE}%MKUKATPBASIS,%CEXT,%VEXT,%P
EXT  BAS (BAS_COMMAND  :IN,REAL  :IN )
DECL INT SUCCESS
;ENDFOLD (BASISTECH EXT)
;FOLD USER EXT;%{E}%MKUKATPUSER,%CEXT,%VEXT,%P
;Make your modifications here

;ENDFOLD (USER EXT)
;ENDFOLD (EXTERNAL DECLARATIONS)
DECL BASIS_SUGG_T LAST_BASIS={POINT1[] "P_aFOTO1_B2             ",POINT2[] "P_aFOTO1_B2             ",CP_PARAMS[] "CPDAT0                  ",PTP_PARAMS[] "PDAT3                   ",CONT[] "                        ",CP_VEL[] "2.0                     ",PTP_VEL[] "100                     ",SYNC_PARAMS[] "SYNCDAT                 ",SPL_NAME[] "S0                      ",A_PARAMS[] "ADAT0                   "}
DECL PDAT PH={VEL 100.000,ACC 100.000,APO_DIST 100.000,APO_MODE #CDIS,GEAR_JERK 50.0000,EXAX_IGN 0}
DECL PDAT PM={VEL 100.000,ACC 50.0000,APO_DIST 100.000,APO_MODE #CDIS,GEAR_JERK 50.0000,EXAX_IGN 0}
DECL E6POS XP_FOTO1V_Bandeja1={X -1183.89807,Y -595.618103,Z 964.318604,A -96.0049210,B 35.3597450,C 86.8423,S 6,T 58,E1 0.0,E2 0.0,E3 0.0,E4 0.0,E5 0.0,E6 0.0}
DECL FDAT FP_FOTO1V_Bandeja1={TOOL_NO 5,BASE_NO 0,IPO_FRAME #BASE,POINT2[] " ",TQ_STATE FALSE}
DECL E6POS XP_FOTO2V_BANDEJA1={X -993.835266,Y -675.858704,Z 963.521667,A -36.7756958,B 29.1023121,C 104.688148,S 6,T 50,E1 0.0,E2 0.0,E3 0.0,E4 0.0,E5 0.0,E6 0.0}
DECL FDAT FP_FOTO2V_BANDEJA1={TOOL_NO 5,BASE_NO 0,IPO_FRAME #BASE,POINT2[] " ",TQ_STATE FALSE}
DECL E6POS XPOS_ESPERA_FOTO={X -577.117249,Y -209.544479,Z 2331.43652,A -84.9928665,B 10.8814869,C 49.4836502,S 6,T 58,E1 0.0,E2 0.0,E3 0.0,E4 0.0,E5 0.0,E6 0.0}
DECL FDAT FPOS_ESPERA_FOTO={TOOL_NO 5,BASE_NO 0,IPO_FRAME #BASE,POINT2[] " ",TQ_STATE FALSE}
DECL E6POS XP_FOTO1V_Bandeja2={X -1187.09058,Y -744.291260,Z 1047.06836,A -94.8473129,B 36.5673332,C 88.7703781,S 6,T 58,E1 0.0,E2 0.0,E3 0.0,E4 0.0,E5 0.0,E6 0.0}
DECL FDAT FP_FOTO1V_Bandeja2={TOOL_NO 5,BASE_NO 0,IPO_FRAME #BASE,POINT2[] " ",TQ_STATE FALSE}
DECL E6POS XP_FOTO1V_Bandeja3={X -1020.13104,Y -824.657166,Z 1252.74316,A -107.719704,B 35.4580040,C 87.8595428,S 6,T 26,E1 0.0,E2 0.0,E3 0.0,E4 0.0,E5 0.0,E6 0.0}
DECL FDAT FP_FOTO1V_Bandeja3={TOOL_NO 5,BASE_NO 0,IPO_FRAME #BASE,POINT2[] " ",TQ_STATE FALSE}
DECL E6POS XP_FOTO1V_Bandeja4={X -1183.31750,Y -773.952454,Z 1412.69458,A -96.5772705,B 42.2164497,C 85.8641357,S 6,T 26,E1 0.0,E2 0.0,E3 0.0,E4 0.0,E5 0.0,E6 0.0}
DECL FDAT FP_FOTO1V_Bandeja4={TOOL_NO 5,BASE_NO 0,IPO_FRAME #BASE,POINT2[] " ",TQ_STATE FALSE}
DECL E6POS XP_FOTO1V_Bandeja5={X -1183.14099,Y -595.342957,Z 1800.00439,A -95.9583435,B 35.3498039,C 86.8288,S 6,T 26,E1 0.0,E2 0.0,E3 0.0,E4 0.0,E5 0.0,E6 0.0}
DECL FDAT FP_FOTO1V_Bandeja5={TOOL_NO 5,BASE_NO 0,IPO_FRAME #BASE,POINT2[] " ",TQ_STATE FALSE}
DECL E6POS XP_FOTO2V_Bandeja2={X -937.384766,Y -710.244934,Z 879.322144,A -35.2632179,B 29.1483555,C 104.679298,S 6,T 50,E1 0.0,E2 0.0,E3 0.0,E4 0.0,E5 0.0,E6 0.0}
DECL FDAT FP_FOTO2V_Bandeja2={TOOL_NO 5,BASE_NO 0,IPO_FRAME #BASE,POINT2[] " ",TQ_STATE FALSE}
DECL E6POS XP_FOTO2V_Bandeja3={X -993.379395,Y -687.948486,Z 1239.61499,A -36.8665199,B 29.1382885,C 104.710991,S 6,T 50,E1 0.0,E2 0.0,E3 0.0,E4 0.0,E5 0.0,E6 0.0}
DECL FDAT FP_FOTO2V_Bandeja3={TOOL_NO 5,BASE_NO 0,IPO_FRAME #BASE,POINT2[] " ",TQ_STATE FALSE}
DECL E6POS XP_FOTO2V_Bandeja4={X -889.728,Y -700.720154,Z 1428.54895,A -36.8714676,B 29.1350174,C 104.708794,S 6,T 50,E1 0.0,E2 0.0,E3 0.0,E4 0.0,E5 0.0,E6 0.0}
DECL FDAT FP_FOTO2V_Bandeja4={TOOL_NO 5,BASE_NO 0,IPO_FRAME #BASE,POINT2[] " ",TQ_STATE FALSE}
DECL E6POS XP_FOTO2V_Bandeja5={X -993.510437,Y -675.090881,Z 1800.01270,A -36.8860054,B 29.1313248,C 104.699234,S 6,T 50,E1 0.0,E2 0.0,E3 0.0,E4 0.0,E5 0.0,E6 0.0}
DECL FDAT FP_FOTO2V_Bandeja5={TOOL_NO 5,BASE_NO 0,IPO_FRAME #BASE,POINT2[] " ",TQ_STATE FALSE}
DECL LDAT LM={VEL 2.00000,ACC 15.0000,APO_DIST 100.000,APO_FAC 50.0000,AXIS_VEL 100.000,AXIS_ACC 100.000,ORI_TYP #VAR,CIRC_TYP #BASE,JERK_FAC 50.0000,GEAR_JERK 50.0000,EXAX_IGN 0}
DECL E6POS XP10={X -555.796814,Y -30.6566067,Z 2345.89355,A -101.390305,B 10.0001287,C 47.4536476,S 6,T 58,E1 0.0,E2 0.0,E3 0.0,E4 0.0,E5 0.0,E6 0.0}
DECL FDAT FP10={TOOL_NO 5,BASE_NO 0,IPO_FRAME #BASE,POINT2[] " ",TQ_STATE FALSE}
DECL E6POS XP20={X -1201.15967,Y 5.10820818,Z 1800.01270,A -71.3258,B 29.1313248,C 104.699234,S 6,T 26,E1 0.0,E2 0.0,E3 0.0,E4 0.0,E5 0.0,E6 0.0}
DECL FDAT FP20={TOOL_NO 5,BASE_NO 0,IPO_FRAME #BASE,POINT2[] " ",TQ_STATE FALSE}
DECL E6POS XP30={X -52.4755898,Y -328.745148,Z 2555.05981,A -23.5131760,B 6.28098536,C 35.9051781,S 6,T 58,E1 0.0,E2 0.0,E3 0.0,E4 0.0,E5 0.0,E6 0.0}
DECL FDAT FP30={TOOL_NO 5,BASE_NO 0,IPO_FRAME #BASE,POINT2[] " ",TQ_STATE FALSE}
DECL E6POS XP1={X -1182.84875,Y -262.316071,Z 1799.99951,A -95.9618378,B 35.3506813,C 86.8218536,S 6,T 26,E1 0.0,E2 0.0,E3 0.0,E4 0.0,E5 0.0,E6 0.0}
DECL FDAT FP1={TOOL_NO 5,BASE_NO 0,IPO_FRAME #BASE,POINT2[] " ",TQ_STATE FALSE}
DECL E6POS XP_ESPERA_FOTO={X -1182.84875,Y -262.316071,Z 1799.99951,A -95.9618378,B 35.3506813,C 86.8218536,S 6,T 26,E1 0.0,E2 0.0,E3 0.0,E4 0.0,E5 0.0,E6 0.0}
DECL FDAT FP_ESPERA_FOTO={TOOL_NO 5,BASE_NO 0,IPO_FRAME #BASE,POINT2[] " ",TQ_STATE FALSE}
DECL PDAT PPDAT1={VEL 100.000,ACC 100.000,APO_DIST 100.000,GEAR_JERK 50.0000,EXAX_IGN 0}
DECL E6POS XP11={X -577.117249,Y -209.544479,Z 2331.43652,A -84.9928665,B 10.8814869,C 49.4836502,S 6,T 58,E1 0.0,E2 0.0,E3 0.0,E4 0.0,E5 0.0,E6 0.0}
DECL FDAT FP11={TOOL_NO 5,BASE_NO 0,IPO_FRAME #BASE,POINT2[] " ",TQ_STATE FALSE}
DECL E6POS XP2={X -1476.33630,Y 934.788879,Z 2103.11304,A 36.2463837,B -15.5853510,C 56.0520973,S 3,T 42,E1 0.0,E2 0.0,E3 0.0,E4 0.0,E5 0.0,E6 0.0}
DECL FDAT FP2={TOOL_NO 9,BASE_NO 3,IPO_FRAME #BASE,POINT2[] " ",TQ_STATE FALSE}
DECL PDAT PPDAT2={VEL 100.000,ACC 100.000,APO_DIST 100.000,GEAR_JERK 50.0000,EXAX_IGN 0}
DECL E6POS XP_AFOTO1_B2={X -1186.80957,Y -354.904388,Z 1046.96387,A -94.8460388,B 36.5748024,C 88.7817917,S 6,T 58,E1 0.0,E2 0.0,E3 0.0,E4 0.0,E5 0.0,E6 0.0}
DECL FDAT FP_aFOTO1_B2={TOOL_NO 5,BASE_NO 0,IPO_FRAME #BASE,POINT2[] " ",TQ_STATE FALSE}
DECL PDAT PPDAT3={VEL 100.000,ACC 100.000,APO_DIST 100.000,GEAR_JERK 50.0000,EXAX_IGN 0}
ENDDAT
